(* PLC project Unnamed, Unknown Unnamed 1 *)
(* stored: creationDateTime 2026-05-30T20:13:41, modificationDateTime 2026-05-30T20:13:41 *)

PROGRAM main
  VAR
    MainGreen : BOOL := True;
    MainYellow : BOOL := False;
    MainRed : BOOL := False;
    SideGreen : BOOL := False;
    SideYellow : BOOL := False;
    SideRed : BOOL := True;
    CarWaiting : BOOL := False;
    PedWaiting : BOOL := False;
    GreenTimer : TON;
    YellowTimer : TON;
    SideGreenTimer : TON;
    SideYellowTimer : TON;
    SideYeIIowTimer : DINT;
    CycIeActive : BOOL := False;
    CycleActive : BOOL := False;
    TON0 : TON;
  END_VAR

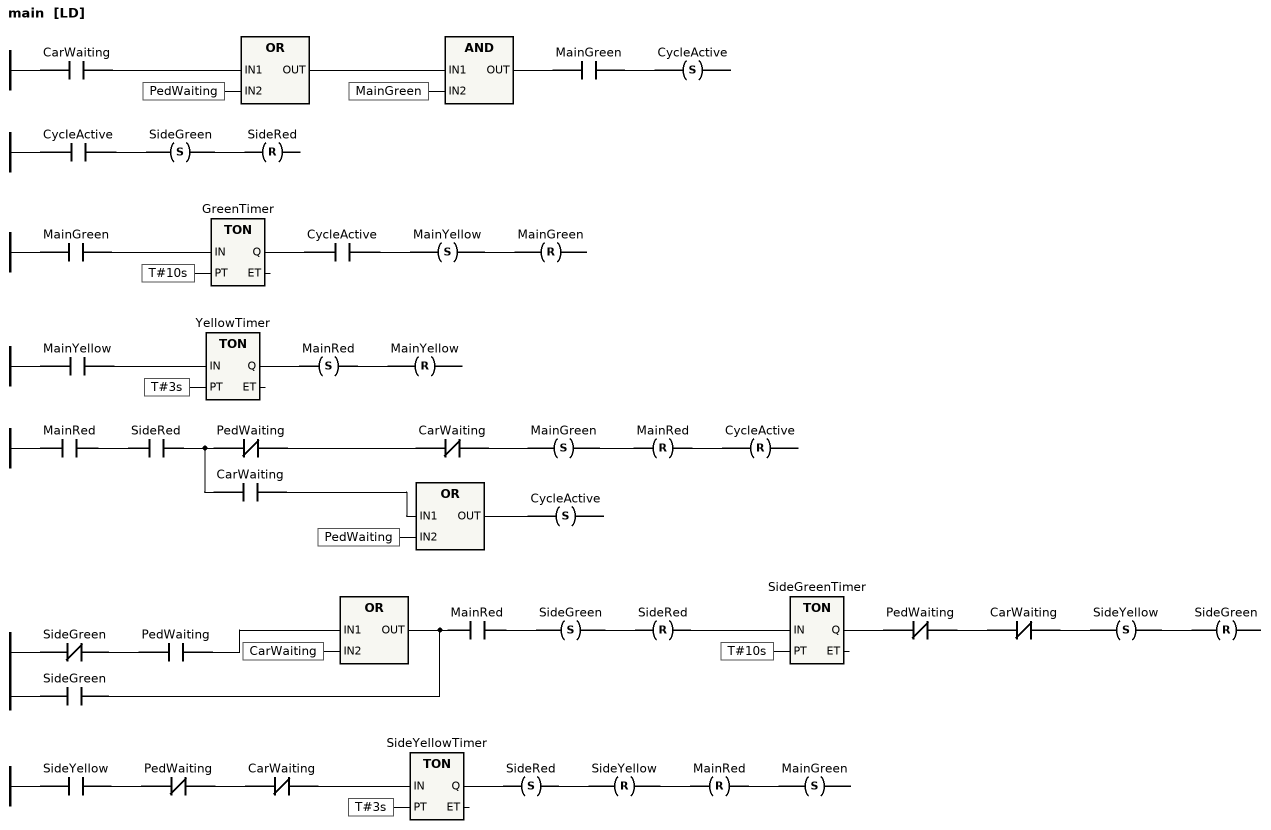
(* LD diagram, written out as Structured Text *)
IF (CarWaiting OR PedWaiting) AND MainGreen AND MainGreen THEN CycleActive := TRUE; END_IF;
IF CycIeActive THEN SideGreen := TRUE; END_IF;
IF CycIeActive THEN SideRed := FALSE; END_IF;
GreenTimer(IN := MainGreen, PT := T#10s);
IF GreenTimer.Q AND CycleActive THEN MainYellow := TRUE; END_IF;
IF GreenTimer.Q AND CycleActive THEN MainGreen := FALSE; END_IF;
YellowTimer(IN := MainYellow, PT := T#3s);
IF YellowTimer.Q THEN MainRed := TRUE; END_IF;
IF YellowTimer.Q THEN MainYellow := FALSE; END_IF;
IF MainRed AND SideRed AND NOT PedWaiting AND NOT CarWaiting THEN MainGreen := TRUE; END_IF;
IF MainRed AND SideRed AND NOT PedWaiting AND NOT CarWaiting THEN MainRed := FALSE; END_IF;
IF MainRed AND SideRed AND NOT PedWaiting AND NOT CarWaiting THEN CycleActive := FALSE; END_IF;
IF MainRed AND SideRed AND CarWaiting OR PedWaiting THEN CycleActive := TRUE; END_IF;
IF (NOT SideGreen AND PedWaiting OR CarWaiting OR SideGreen) AND MainRed THEN SideGreen := TRUE; END_IF;
IF (NOT SideGreen AND PedWaiting OR CarWaiting OR SideGreen) AND MainRed THEN SideRed := FALSE; END_IF;
SideGreenTimer(IN := (NOT SideGreen AND PedWaiting OR CarWaiting OR SideGreen) AND MainRed, PT := T#10s);
IF SideGreenTimer.Q AND NOT PedWaiting AND NOT CarWaiting THEN SideYellow := TRUE; END_IF;
IF SideGreenTimer.Q AND NOT PedWaiting AND NOT CarWaiting THEN SideGreen := FALSE; END_IF;
SideYellowTimer(IN := SideYellow AND NOT PedWaiting AND NOT CarWaiting, PT := T#3s);
IF SideYellowTimer.Q THEN SideRed := TRUE; END_IF;
IF SideYellowTimer.Q THEN SideYellow := FALSE; END_IF;
IF SideYellowTimer.Q THEN MainRed := FALSE; END_IF;
IF SideYellowTimer.Q THEN MainGreen := TRUE; END_IF;
END_PROGRAM

CONFIGURATION Config0
  RESOURCE Res0 ON PLC
    TASK task0(INTERVAL := T#20ms, PRIORITY := 1);
    PROGRAM instance0 WITH task0 : main;
  END_RESOURCE
END_CONFIGURATION
